// TIA Portal V19 export
FUNCTION "MwFakCalc_CALL" : Void   // FC177, LAD
TITLE = MW FAK CALC CALL
// stored: SetENOAutomatically false
BEGIN

REGION Network 1: Data In - PB Push Ax
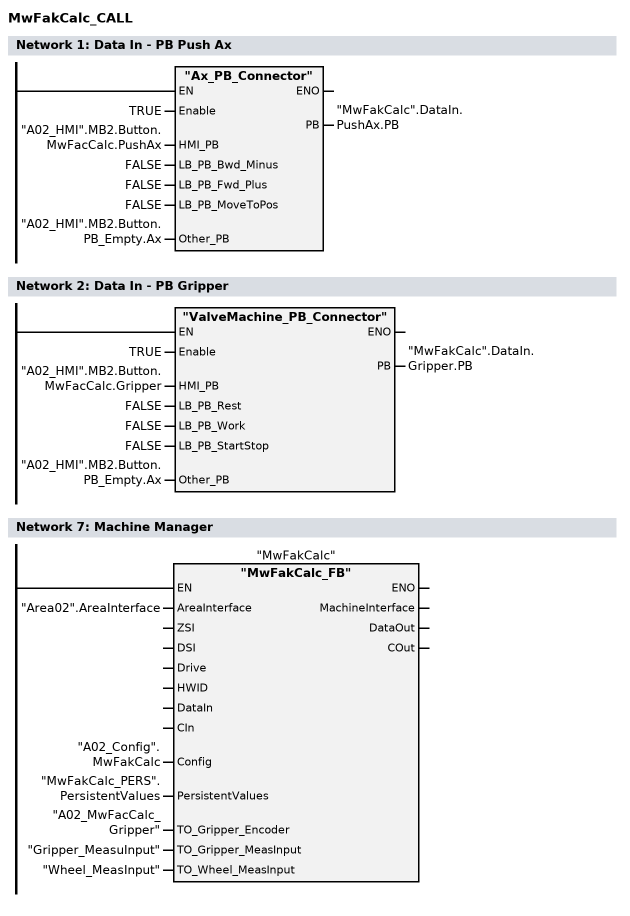
   RUNG wire#powerrail
      "Ax_PB_Connector"(Enable := TRUE, HMI_PB := "A02_HMI".MB2.Button.MwFacCalc.PushAx, LB_PB_Bwd_Minus := FALSE, LB_PB_Fwd_Plus := FALSE, LB_PB_MoveToPos := FALSE, Other_PB := "A02_HMI".MB2.Button.PB_Empty.Ax, PB => "MwFakCalc".DataIn.PushAx.PB)
   END_RUNG
   // the same network as SCL:
   "Ax_PB_Connector"(Enable := TRUE,
                     HMI_PB := "A02_HMI".MB2.Button.MwFacCalc.PushAx,
                     LB_PB_Bwd_Minus := FALSE,
                     LB_PB_Fwd_Plus := FALSE,
                     LB_PB_MoveToPos := FALSE,
                     Other_PB := "A02_HMI".MB2.Button.PB_Empty.Ax,
                     PB => "MwFakCalc".DataIn.PushAx.PB);
END_REGION

REGION Network 2: Data In - PB Gripper
   RUNG wire#powerrail
      "ValveMachine_PB_Connector"(Enable := TRUE, HMI_PB := "A02_HMI".MB2.Button.MwFacCalc.Gripper, LB_PB_Rest := FALSE, LB_PB_Work := FALSE, LB_PB_StartStop := FALSE, Other_PB := "A02_HMI".MB2.Button.PB_Empty.Ax, PB => "MwFakCalc".DataIn.Gripper.PB)
   END_RUNG
   // the same network as SCL:
   "ValveMachine_PB_Connector"(Enable := TRUE,
                           HMI_PB := "A02_HMI".MB2.Button.MwFacCalc.Gripper,
                           LB_PB_Rest := FALSE,
                           LB_PB_Work := FALSE,
                           LB_PB_StartStop := FALSE,
                           Other_PB := "A02_HMI".MB2.Button.PB_Empty.Ax,
                           PB => "MwFakCalc".DataIn.Gripper.PB);
END_REGION

REGION Network 3 (SCL): DataIn - Sensor
   "MwFakCalc".DataIn.MaterialPresenceEntry := "A0201_Carrello_Riposizionatore_Phc_Prima_Encoder" OR "A0201_Profila_Phc_Prima_Encoder" OR "A02_DEBUG".MatPresence_AfterMW;
   "MwFakCalc".DataIn.MaterialPresenceExit := "A0201_Carrello_Riposizionatore_Phc_Dopo_Encoder" OR "A02_DEBUG".MatPresence_AfterFAK;
   "MwFakCalc".DataIn.MaterialJam := "A0201_Ls_Controllo_Inceppamento";

   "MwFakCalc".DataIn.PushAx_Ls_HomeFwd := "A0201_Carrello_Misuratore_Posizione_Zero";
   "MwFakCalc".DataIn.PushAx_Ls_RestBwd := "A0201_Carrello_Misuratore_Stop_Verso_Rest";
   "MwFakCalc".DataIn.PushAx_Ls_LowSpeedHome := "A0201_Carrello_Misuratore_Rallentamento_Verso_Zero";
   "MwFakCalc".DataIn.PushAx_Ls_LowSpeedRest := "A0201_Carrello_Misuratore_Rallentamento_Verso_Posizione_Rest"; 
   "MwFakCalc".DataIn.PushAx_Ls_Touch := "A0201_Carrello_Misuratore_In_Appoggio_Tra_Loro";
   "MwFakCalc".DataIn.Gripper_Ls_ForceOpen := "A0201_Carrello_Misuratore_Posizione_Work";

   "MwFakCalc".DataIn.Gripper.Rest_Ls[1] := "A0201_Pinza_Misuratore_Ls_Rest";
   "MwFakCalc".DataIn.Gripper.Work_Ls[1] := "A0201_Pinza_Misuratore_Ls_Work";
END_REGION

REGION Network 4 (SCL): Safety

   "MwFakCalc".ZSI := "F_DB".ZSI_Zone13;

   "MwFakCalc".DSI.PushAx := "F_DB".DSI_S120_FAK_Pusher;

   "MwFakCalc".DSI.Gripper := "F_DB".DSI_V_Air_A0301_A0302;
END_REGION

REGION Network 5 (SCL): Drive e HWID

   "MwFakCalc".Drive.PushAx.Infeed_ON := "Areas_ITF".AG.Infeed_Running;
   "MwFakCalc".Drive.PushAx.AccessPoint := "HW_Const_Values".CU3_PROFINET_interface_590A1_ModuleAccessPoint;
   "MwFakCalc".Drive.PushAx.AxisID := "CU3_ID_6_1260A1_1_1260M1";
   "MwFakCalc".Drive.PushAx.TokenChain := "TOKENCHAIN_CU3";


   "MwFakCalc".HWID.PushAx_TEL1 := "HW_Const_Values".CU3_PROFINET_interface_1260A1_1_Standard_telegram_1;
END_REGION

REGION Network 6 (SCL): Cin
   "MwFakCalc".CIn.Manager.EnableStopDoorOpeningReq := TRUE;
   "MwFakCalc".CIn.Manager.EnableStopInPhase := "RollformingMng".MachineInterface.AckStopInPhase;
   "MwFakCalc".CIn.Manager.EnableStopProgrammed := "RollformingMng".MachineInterface.AckStopProgrammed;


   "MwFakCalc".CIn.Rollformer_Standstill := "Rollformer".COut.Feed.Standstill;
   "MwFakCalc".CIn.Rollformer_CheckNextFwd := "Rollformer".COut.Feed.Fwd_CheckNext;
   "MwFakCalc".CIn.Rollformer_CheckNextBwd := "Rollformer".COut.Feed.Bwd_CheckNext;

   "MwFakCalc".CIn.MW_ActualFAK := "PostPunchingMatCounter_PERS".PersistentValues.Data.FAK;

   "MwFakCalc".CIn.SemiAut_And_ButtonPressed := "RollformingMng".Sts.Semiautomatic;

   "MwFakCalc".CIn.PostServo_MeasuredID := "MwFakCalc_PS".MeasureID;
   "MwFakCalc".CIn.PostServo_MeasuredValueG := "MwFakCalc_PS".MeasuredValueG;
   "MwFakCalc".CIn.PostServo_MeasuredValueW := "MwFakCalc_PS".MeasuredValueW;
END_REGION

REGION Network 7: Machine Manager
   RUNG wire#powerrail
      "MwFakCalc"(AreaInterface := "Area02".AreaInterface, ZSI :=, DSI :=, Drive :=, HWID :=, DataIn :=, CIn :=, Config := "A02_Config".MwFakCalc, PersistentValues := "MwFakCalc_PERS".PersistentValues, TO_Gripper_Encoder := "A02_MwFacCalc_Gripper", TO_Gripper_MeasInput := "Gripper_MeasuInput", TO_Wheel_MeasInput := "Wheel_MeasInput", MachineInterface =>, DataOut =>, COut =>)
   END_RUNG
   // the same network as SCL:
   "MwFakCalc"(AreaInterface := "Area02".AreaInterface,   // "MwFakCalc_FB"
               Config := "A02_Config".MwFakCalc,
               PersistentValues := "MwFakCalc_PERS".PersistentValues,
               TO_Gripper_Encoder := "A02_MwFacCalc_Gripper",
               TO_Gripper_MeasInput := "Gripper_MeasuInput",
               TO_Wheel_MeasInput := "Wheel_MeasInput");
END_REGION

REGION Network 8 (SCL): Data Out
   "A0201_Pinza_Misuratore_V_Rest" := "MwFakCalc".DataOut.Gripper.RestSolenoid;
   "A0201_Pinza_Misuratore_V_Work" := "MwFakCalc".DataOut.Gripper.WorkSolenoid;

   "CU320_Trigger_Lettura_Correzione_Encoder" := "MwFakCalc".DataOut.MeasInput_ExeReg;
   "MwFakCalc_PS".StartMeasure :="MwFakCalc".DataOut.MeasInput_ExeReg;
END_REGION

REGION Network 9: >
END_REGION
END_FUNCTION
